INTERFACE ITF_Communicator EXTENDS ITF_MessengerSender, ITF_MessengerRecipient

END_INTERFACE

(* stored: Version 1.1.0.1
   Itf ITF_Communicator: Id {95c8f21f-348b-0804-2e77-1d9f40277cd9} *)
